# EPICS substitutions: db/Beckhoff_4XXX/ecmcEL4122.substitutions
#4..20mA (0..32767)
file "ecmc_analogOutput-chX.template"
{
  pattern {CH_ID, ESLO, EOFF, EGU, PREC, LOW, LOLO, HIGH, HIHI, HYST, LLSV, LSV, HSV, HHSV, DRVL, DRVH}
          {01, "${_ESLO=4.882961516E-4}", "${_EOFF=4}", "${_EGU=mA}", "${_PREC=3}", 4, 3.9, 20, 20.1, 0, "MAJOR", "MINOR", "MINOR", "MAJOR", 4, 20}
          {02, "${_ESLO=4.882961516E-4}", "${_EOFF=4}", "${_EGU=mA}", "${_PREC=3}", 4, 3.9, 20, 20.1, 0, "MAJOR", "MINOR", "MINOR", "MAJOR", 4, 20}
}
